TYPE (* A Template for a Data Type *)
  (* Version 1.0, 2024-12-18, cochicde *)
  PACKAGE performance;
  MyStruct : STRUCT
    _int : INT;
    _string : STRING;
  END_STRUCT;
END_TYPE
